// TIA Portal V16 export
// export: Created 2022-09-01T14:27:09.4933428Z, ExportSetting WithDefaults, DisplayName Totally Integrated Automation Portal, DisplayVersion V16, DisplayName TIA Portal Version Control Interface, DisplayVersion V16, DisplayName TIA Portal Openness, DisplayVersion V16, DisplayName STEP 7 Professional, DisplayVersion V16, DisplayName STEP 7 Safety, DisplayVersion V16, DisplayName WinCC Advanced, DisplayVersion V16
VAR_GLOBAL   // PLC tag table "Inputs"
   "EV1.1_ABERTA" AT %I0.0 : Bool;
   "EV1.1_FECHADA" AT %I0.1 : Bool;
   "EV2.1_ABERTA" AT %I0.2 : Bool;
   "EV2.1_FECHADA" AT %I0.3 : Bool;
   "EV3.1_ABERTA" AT %I0.4 : Bool;
   "EV3.1_FECHADA" AT %I0.5 : Bool;
   "EV4.1_ABERTA" AT %I0.6 : Bool;
   "EV4.1_FECHADA" AT %I0.7 : Bool;
   "EV5.1_ABERTA" AT %I1.0 : Bool;
   "EV5.1_FECHADA" AT %I1.1 : Bool;
   "EV1.2_ABERTA" AT %I1.2 : Bool;
   "EV1.2_FECHADA" AT %I1.3 : Bool;
   "EV2.2_ABERTA" AT %I1.4 : Bool;
   "EV2.2_FECHADA" AT %I1.5 : Bool;
   "EV3.2_ABERTA" AT %I2.0 : Bool;
   "EV3.2_FECHADA" AT %I2.1 : Bool;
   "EV4.2_ABERTA" AT %I2.2 : Bool;
   "EV4.2_FECHADA" AT %I2.3 : Bool;
   "EV5.2_ABERTA" AT %I2.4 : Bool;
   "EV5.2_FECHADA" AT %I2.5 : Bool;
   PRESSOSTATO_1 AT %IW4 : Word;
   PRESSOSTATO_2 AT %IW6 : Word;
   AVARIA_BOMBA_1 AT %I2.6 : Bool;
   AVARIA_BOMBA_2 AT %I2.7 : Bool;
   AVARIA_BOMBA_3 AT %I3.0 : Bool;
END_VAR
